FUNCTION_BLOCK ROBOT7TESTFB (* JADE WORKER *)
  (* Standard: 61499-1 *)
  (* Version 1.0, 2014-04-22, Ahmed, Fraunhofer IGD *)
  (* Compiler header: package fb.rt; *)
  (* Compiler Java Sun JDK 1.5.0 *)
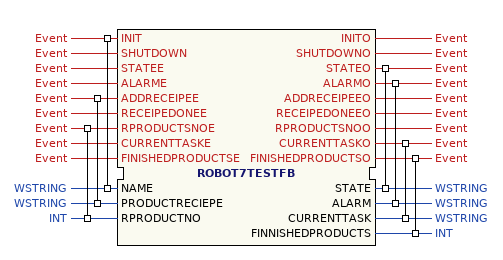
  EVENT_INPUT
    INIT WITH NAME; (* Normal Execution Request *)
    SHUTDOWN;
    STATEE;
    ALARME;
    ADDRECEIPEE WITH PRODUCTRECIEPE; (* Normal Execution Request *)
    RECEIPEDONEE;
    RPRODUCTSNOE WITH RPRODUCTNO;
    CURRENTTASKE;
    FINISHEDPRODUCTSE;
  END_EVENT
  EVENT_OUTPUT
    INITO; (* Execution Confirmation *)
    SHUTDOWNO;
    STATEO WITH STATE;
    ALARMO WITH ALARM;
    ADDRECEIPEEO; (* Execution Confirmation *)
    RECEIPEDONEEO;
    RPRODUCTSNOO;
    CURRENTTASKO WITH CURRENTTASK;
    FINISHEDPRODUCTSO WITH FINNISHEDPRODUCTS;
  END_EVENT
  VAR_INPUT
    NAME : WSTRING;
    PRODUCTRECIEPE : WSTRING;
    RPRODUCTNO : INT;
  END_VAR
  VAR_OUTPUT
    STATE : WSTRING;
    ALARM : WSTRING;
    CURRENTTASK : WSTRING;
    FINNISHEDPRODUCTS : INT;
  END_VAR
END_FUNCTION_BLOCK
